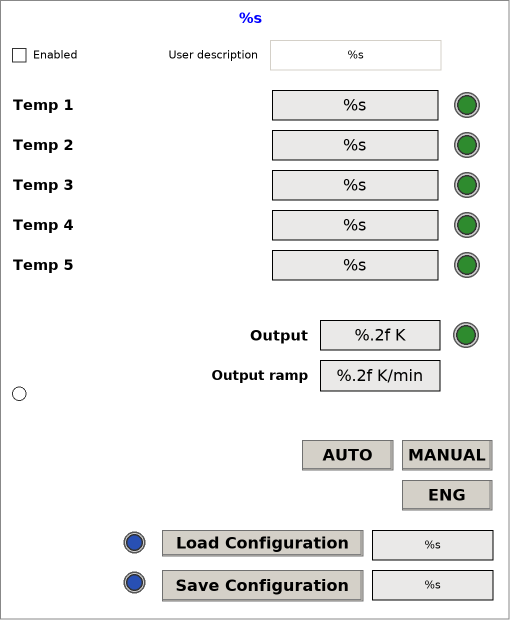
VISUALIZATION TEMPLATE_TEMPERATURE_VOTE  // 510x620
VAR_IN_OUT
	m_Instance : FB_METIS_VOTER; 
	m_all_temperatures_array: FB_METIS_TEMPERATURES;
END_VAR
    Rectangle (10,3 481x30), "%s", tooltip "vote Temperature", text variable: m_Instance.in_sName
    Rectangle (10,90 68x30), "Temp 1"
    Rectangle (10,130 68x30), "Temp 2"
    Rectangle (10,170 68x30), "Temp 3"
    Rectangle (10,210 68x30), "Temp 4"
    Rectangle (10,250 68x30), "Temp 5"
    Lamp1 (452,90 30x30), variable: m_Instance.aTempPointers[0]^.stat.bValid, style: Lamp-Lamp1-Green
    Lamp1 (452,130 30x30), variable: m_Instance.aTempPointers[1]^.stat.bValid, style: Lamp-Lamp1-Green
    Lamp1 (452,170 30x30), variable: m_Instance.aTempPointers[2]^.stat.bValid, style: Lamp-Lamp1-Green
    Lamp1 (452,210 30x30), variable: m_Instance.aTempPointers[3]^.stat.bValid, style: Lamp-Lamp1-Green
    Lamp1 (452,250 30x30), variable: m_Instance.aTempPointers[4]^.stat.bValid, style: Lamp-Lamp1-Green
    RadioButton (10,306 162x175), variable: m_Instance.stat.nVoteMethod, input disabled if: NOT m_Instance.bEngMode
        Areas[0]: Text=Lowest Temperature
        Areas[1]: Text=Highest Temperature
        Areas[2]: Text=Average
        Areas[3]: Text=First Valid
        p340057476: Lowest Temperature
        p3123465237: Highest Temperature
        p2481256679: Average
        p1032612214: First Valid
        p3228930307: Median
        p1847394450: Temperature 2oo3
        p1205187680: Temperature 3oo5
    Rectangle (320,320 120x30), "%.2f K", tooltip "Voting Temperature out [K]", text variable: m_instance.stat.lrTempK
    Lamp1 (451,320 30x30), variable: m_Instance.stat.bValid, style: Lamp-Lamp1-Green
    Rectangle (272,90 166x30), "%s", tooltip "Voting Temperature out [K]", text variable: m_Instance.aTempPointers[0]^.stat.sName
    Rectangle (272,130 166x30), "%s", tooltip "Voting Temperature out [K]", text variable: m_Instance.aTempPointers[1]^.stat.sName
    Rectangle (272,170 166x30), "%s", tooltip "Voting Temperature out [K]", text variable: m_Instance.aTempPointers[2]^.stat.sName
    Rectangle (272,210 166x30), "%s", tooltip "Voting Temperature out [K]", text variable: m_Instance.aTempPointers[3]^.stat.sName
    Rectangle (272,250 166x30), "%s", tooltip "Voting Temperature out [K]", text variable: m_Instance.aTempPointers[4]^.stat.sName
    Button (302,440 91x30), "AUTO", tooltip "Switch to AUTO Mode", colour toggle: m_instance.bAutoMode, input disabled if: m_instance.bAutoMode OR m_instance.bEngMode
        OnMouseClick: execute { m_instance.bAutoMode := TRUE; m_instance.bPLC_HMI := FALSE; }
    Button (402,480 90x30), "ENG", tooltip "Toggle Engineering Mode", colour toggle: m_instance.bEngMode, input disabled if: m_instance.bAutoMode
        toggle m_instance.bEngMode
    Button (402,440 90x30), "MANUAL", tooltip "Switch to MANUAL Mode", colour toggle: NOT m_instance.bAutoMode, input disabled if: NOT m_instance.bAutoMode AND NOT m_instance.bEngMode
        OnMouseClick: execute {
            m_instance.bAutoMode := FALSE;
            m_instance.bManualMode := TRUE;
            m_instance.bPLC_HMI := TRUE;
        }
    Lamp1 (122,530 25x25), tooltip "Command coming from the Control System", variable: m_instance.bReadConfig, style: Lamp-Lamp1-Blue
    Button (162,570 201x31), "Save Configuration", input disabled if: NOT m_instance.bEngMode
        OnMouseClick: execute { m_instance.bWriteConfig := TRUE; }
    Button (162,530 201x26), "Load Configuration", input disabled if: NOT m_instance.bEngMode
        OnMouseClick: execute { m_instance.bReadConfig := TRUE; }
    Lamp1 (122,570 25x25), tooltip "Command coming from the Control System", variable: m_instance.bWriteConfig, style: Lamp-Lamp1-Blue
    Rectangle (320,360 120x31), "%.2f K/min", tooltip "Ramp [K/min]", text variable: m_instance.stat.lrRamp
    Rectangle (372,530 121x30), "%s", text variable: m_Instance.fbTempVoteConfig.sReadError, colour toggle: m_Instance.fbTempVoteConfig.bReadError
    Rectangle (372,570 121x30), "%s", text variable: m_Instance.fbTempVoteConfig.sWriteError, colour toggle: m_Instance.fbTempVoteConfig.bWriteError
    Checkbox (10,40 111x30), "Enabled", variable: m_Instance.stat.bEnabled, input disabled if: NOT m_Instance.bEngMode
    Label (110,40 151x30), "User description"
    Textfield (270,40 171x30), "%s", text variable: m_Instance.stat.sDescription, input disabled if: NOT m_Instance.bEngMode
        OnMouseClick: write the text variable via Default
    Rectangle (210,320 101x31), "Output"
    Rectangle (210,360 101x31), "Output ramp"
END_VISUALIZATION

// HMI/VISUs/Util/Button/VISU_HMI_ROUTINES_BUTTON
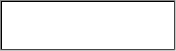
VISUALIZATION VISU_HMI_ROUTINES_BUTTON  // 176x51
VAR_IN_OUT
    m_Hmi : FB_HMI_BUTTON;
END_VAR
    Rectangle (0,0 175x50), invisible if: m_Hmi.bIsNotOrange
    Rectangle (0,0 175x50), invisible if: m_Hmi.bIsNotGray
    Rectangle (0,0 175x50), invisible if: m_Hmi.bIsNotBlue
    Rectangle (0,0 175x50), invisible if: m_Hmi.bIsNotRed
    Rectangle (0,0 175x50), invisible if: m_Hmi.bIsNotGreen
    Rectangle (0,0 175x50), "%s", text variable: m_Hmi.sName
    Rectangle (0,0 175x50), invisible if: m_Hmi.bNotActivated
    Line (0,49) (175,49), invisible if: m_Hmi.bActivated
    Line (174,0) (174,50), invisible if: m_Hmi.bActivated
    Line (174,0) (0,0), invisible if: m_Hmi.bActivated
    Line (0,49) (0,0), invisible if: m_Hmi.bActivated
    Line (175,50) (175,1), invisible if: m_Hmi.bNotActivated
    Line (0,1) (174,1), invisible if: m_Hmi.bNotActivated
    Line (1,0) (1,49), invisible if: m_Hmi.bNotActivated
    Line (175,50) (1,50), invisible if: m_Hmi.bNotActivated
END_VISUALIZATION

// HMI/VISUs/Util/Button/VISU_HMI_SUBSUBSYSTEM_BUTTON
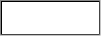
VISUALIZATION VISU_HMI_SUBSUBSYSTEM_BUTTON  // 101x36
VAR_IN_OUT
    m_Hmi : FB_HMI_BUTTON;
END_VAR
    Rectangle (0,0 100x35), invisible if: m_Hmi.bIsNotOrange
    Rectangle (0,0 100x35), invisible if: m_Hmi.bIsNotGray
    Rectangle (0,0 100x35), invisible if: m_Hmi.bIsNotBlue
    Rectangle (0,0 100x35), invisible if: m_Hmi.bIsNotRed
    Rectangle (0,0 100x35), invisible if: m_Hmi.bIsNotGreen
    Rectangle (0,0 100x35), "%s", text variable: m_Hmi.sName
    Rectangle (0,0 100x35), invisible if: m_Hmi.bNotActivated
    Line (0,34) (100,34), invisible if: m_Hmi.bActivated
    Line (99,0) (99,35), invisible if: m_Hmi.bActivated
    Line (98,0) (0,0), invisible if: m_Hmi.bActivated
    Line (0,35) (0,0), invisible if: m_Hmi.bActivated
    Line (100,35) (100,1), invisible if: m_Hmi.bNotActivated
    Line (0,1) (99,1), invisible if: m_Hmi.bNotActivated
    Line (1,0) (1,35), invisible if: m_Hmi.bNotActivated
    Line (100,35) (1,35), invisible if: m_Hmi.bNotActivated
END_VISUALIZATION

// HMI/VISUs/Util/Button/VISU_HMI_SUBSYSTEM_BUTTON
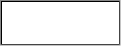
VISUALIZATION VISU_HMI_SUBSYSTEM_BUTTON  // 121x46
VAR_IN_OUT
    m_Hmi : FB_HMI_BUTTON;
END_VAR
    Rectangle (0,0 120x45), invisible if: m_Hmi.bIsNotOrange
    Rectangle (0,0 120x45), invisible if: m_Hmi.bIsNotGray
    Rectangle (0,0 120x45), invisible if: m_Hmi.bIsNotBlue
    Rectangle (0,0 120x45), invisible if: m_Hmi.bIsNotRed
    Rectangle (0,0 120x45), invisible if: m_Hmi.bIsNotGreen
    Rectangle (0,0 120x45), "%s", text variable: m_Hmi.sName
    Rectangle (0,0 120x45), invisible if: m_Hmi.bNotActivated
    Line (0,44) (120,44), invisible if: m_Hmi.bActivated
    Line (119,0) (119,45), invisible if: m_Hmi.bActivated
    Line (118,0) (0,0), invisible if: m_Hmi.bActivated
    Line (0,45) (0,0), invisible if: m_Hmi.bActivated
    Line (120,45) (120,1), invisible if: m_Hmi.bNotActivated
    Line (0,1) (119,1), invisible if: m_Hmi.bNotActivated
    Line (1,0) (1,45), invisible if: m_Hmi.bNotActivated
    Line (120,45) (1,45), invisible if: m_Hmi.bNotActivated
END_VISUALIZATION

// HMI/VISUs/Util/Button/VISU_HMI_SYSTEM_BUTTON
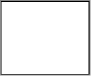
VISUALIZATION VISU_HMI_SYSTEM_BUTTON  // 91x76
VAR_IN_OUT
    m_Hmi : FB_HMI_BUTTON;
END_VAR
    Rectangle (0,0 90x75), invisible if: m_Hmi.bIsNotOrange
    Rectangle (0,0 90x75), invisible if: m_Hmi.bIsNotGray
    Rectangle (0,0 90x75), invisible if: m_Hmi.bIsNotBlue
    Rectangle (0,0 90x75), invisible if: m_Hmi.bIsNotRed
    Rectangle (0,0 90x75), invisible if: m_Hmi.bIsNotGreen
    Rectangle (0,50 90x25), "%s", text variable: m_Hmi.sName
    Image (25,10 40x40), image: VISU_HMI_BUTTON_IMAGES.Start
        p84334746: m_Hmi.sIconName
    Rectangle (0,0 90x75), invisible if: m_Hmi.bNotActivated
    Line (0,74) (90,74), invisible if: m_Hmi.bActivated
    Line (89,75) (89,0), invisible if: m_Hmi.bActivated
    Line (0,74) (0,0), invisible if: m_Hmi.bActivated
    Line (88,0) (0,0), invisible if: m_Hmi.bActivated
    Line (0,1) (90,1), invisible if: m_Hmi.bNotActivated
    Line (1,75) (1,0), invisible if: m_Hmi.bNotActivated
    Line (90,75) (1,75), invisible if: m_Hmi.bNotActivated
    Line (90,75) (90,1), invisible if: m_Hmi.bNotActivated
END_VISUALIZATION

// HMI/VISU_HMI
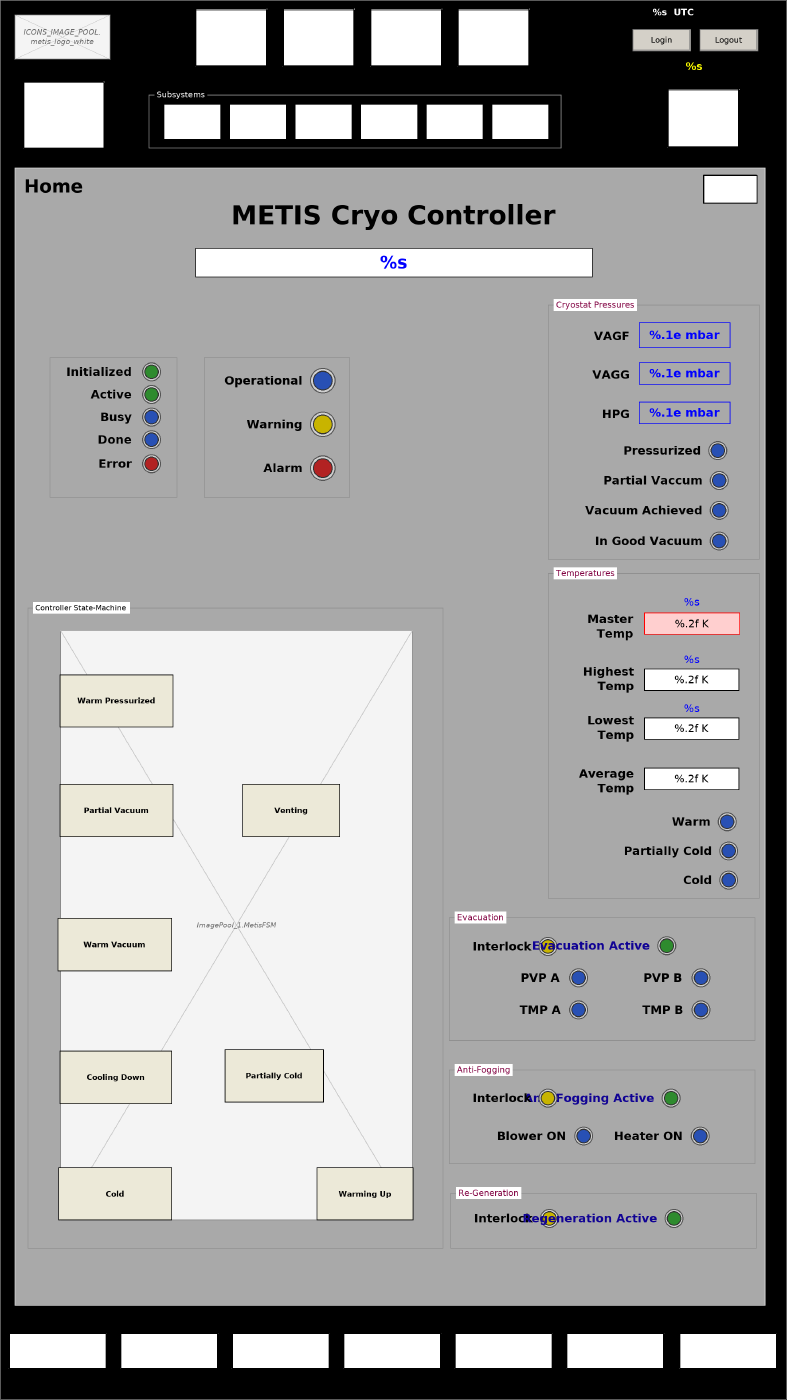
VISUALIZATION VISU_HMI  // 1080x1920
    Frame (388,12 100x80)
        shows VISU_HMI_SYSTEM_BUTTON(m_Hmi := PRG_HMI.fbServicesButton)
        OnMouseClick: execute { PRG_HMI.eActiveTab := E_HMI_TABS.SERVICES; }
    Frame (268,12 100x80)
        shows VISU_HMI_SYSTEM_BUTTON(m_Hmi := PRG_HMI.fbHomeButton)
        OnMouseClick: execute { PRG_HMI.eActiveTab := E_HMI_TABS.HOME; }
    Rectangle (20,230 1030x1560)
    Frame (20,230 1030x1560), frame switch variable: PRG_HMI.eActiveTab
        shows VISU_HMI_HOME(m_instance := MAIN.met_cryo_ctrl)
        shows VISU_HMI_SERVICES()
        shows VISU_HMI_EVACUATION()
        shows VISU_HMI_COOL_DOWN(m_instance := MAIN.met_cryo_ctrl.met_cool_down, m_Cry_Instance := MAIN.met_cryo_ctrl)
        shows VISU_HMI_WARM_UP(m_instance := MAIN.met_cryo_ctrl.met_warm_up, m_Cry_Instance := MAIN.met_cryo_ctrl)
        shows VISU_HMI_VENTING(m_instance := MAIN.met_cryo_ctrl.met_venting, m_Cry_Instance := MAIN.met_cryo_ctrl)
        shows VISU_HMI_ANTI_FOGGING(m_instance := MAIN.met_cryo_ctrl.met_anti_fogging)
        shows VISU_HMI_REGENERATION(m_instance := MAIN.met_cryo_ctrl.met_regeneration)
        shows VISU_HMI_POWER_OUTAGE()
        shows VISU_HMI_CABINETS()
        shows VISU_HMI_VALVES()
        shows VISU_HMI_CONTROL_UNITS()
        shows VISU_HMI_CRY(met_cryo_ctrl := MAIN.met_cryo_ctrl, m_Hmi := PRG_HMI.fbCry)
        shows VISU_HMI_CFO()
        shows VISU_HMI_IMG(m_Temperatures := MAIN.met_cryo_ctrl.met_temp, m_Voters := MAIN.met_cryo_ctrl.met_voters, m_Tctrl := MAIN.met_cryo_ctrl.met_tctrl, m_Heaters := MAIN.met_cryo_ctrl.met_heaters, m_Lakeshores := MAIN.met_cryo_ctrl.met_lakeshores, m_Hmi := PRG_HMI.fbImg)
        shows VISU_HMI_LMS()
        shows VISU_HMI_SCA(m_Temperatures := MAIN.met_cryo_ctrl.met_temp, m_Voters := MAIN.met_cryo_ctrl.met_voters, m_Tctrl := MAIN.met_cryo_ctrl.met_tctrl, m_Heaters := MAIN.met_cryo_ctrl.met_heaters, m_Lakeshores := MAIN.met_cryo_ctrl.met_lakeshores, m_Hmi := PRG_HMI.fbSca)
        shows VISU_HMI_ICS(m_CCUs := MAIN.met_cryo_ctrl.met_ccus, m_Hmi := PRG_HMI.fbIcs)
        shows VISU_HMI_HEATERS()
        shows VISU_HMI_EVENTS()
        shows VISU_HMI_PRESSURES()
        shows VISU_HMI_COOLERS()
        shows VISU_HMI_PUMPS(m_Hmi := PRG_HMI.fbPumps)
        shows VISU_HMI_TEMPERATURES(met_cryo_ctrl := MAIN.met_cryo_ctrl, m_Hmi := PRG_HMI.fbTemperatures)
        shows VISU_HMI_ICS_INTERLOCKS()
        shows VISU_HMI_DETECTORS()
        shows VISU_HMI_CONTROL_LOOPS()
        shows VISU_SIM_PRESS_AND_TEMPS()
        pReferences[1]: m_Instance=MAIN.fbServices, m_Hmi=PRG_HMI.fbServices
        p1199675002: PRG_HMI.fbSca
        p3123483648: PRG_HMI.fbPumps
        p2939190159: MAIN.met_cryo_ctrl
    Image (20,20 131x61), image: ICONS_IMAGE_POOL.metis_logo_white
    Rectangle (774,4 300x25), "%s UTC", text variable: MAIN.met_cryo_ctrl.met_cry_time.stat.sUtcTime
    Frame (12,1828 135x50)
        shows VISU_HMI_ROUTINES_BUTTON(m_Hmi := PRG_HMI.fbEvacuationButton)
        OnMouseClick: execute { PRG_HMI.eActiveTab := E_HMI_TABS.EVACUATION; }
    Frame (165,1828 135x50)
        shows VISU_HMI_ROUTINES_BUTTON(m_Hmi := PRG_HMI.fbCoolDownButton)
        OnMouseClick: execute { PRG_HMI.eActiveTab := E_HMI_TABS.COOL_DOWN; }
    Frame (318,1828 135x50)
        shows VISU_HMI_ROUTINES_BUTTON(m_Hmi := PRG_HMI.fbWarmUpButton)
        OnMouseClick: execute { PRG_HMI.eActiveTab := E_HMI_TABS.WARM_UP; }
    Frame (471,1828 135x50)
        shows VISU_HMI_ROUTINES_BUTTON(m_Hmi := PRG_HMI.fbVentingButton)
        OnMouseClick: execute { PRG_HMI.eActiveTab := E_HMI_TABS.VENTING; }
    Frame (624,1828 135x50)
        shows VISU_HMI_ROUTINES_BUTTON(m_Hmi := PRG_HMI.fbRegenerationButton)
        OnMouseClick: execute { PRG_HMI.eActiveTab := E_HMI_TABS.REGENERATION; }
    Frame (777,1828 135x50)
        shows VISU_HMI_ROUTINES_BUTTON(m_Hmi := PRG_HMI.fbAntiFoggingButton)
        OnMouseClick: execute { PRG_HMI.eActiveTab := E_HMI_TABS.ANTI_FOGGING; }
    Frame (932,1828 135x50)
        shows VISU_HMI_ROUTINES_BUTTON(m_Hmi := PRG_HMI.fbPowerOutageButton)
        OnMouseClick: execute { PRG_HMI.eActiveTab := E_HMI_TABS.POWER_OUTAGE; }
    Frame (508,12 100x80)
        shows VISU_HMI_SYSTEM_BUTTON(m_Hmi := PRG_HMI.fbEventsButton)
        OnMouseClick: execute { PRG_HMI.eActiveTab := E_HMI_TABS.EVENTS; }
    Frame (628,12 100x80)
        shows VISU_HMI_SYSTEM_BUTTON(m_Hmi := PRG_HMI.fbIcsInterlocksButton)
        OnMouseClick: execute { PRG_HMI.eActiveTab := E_HMI_TABS.ICS_INTERLOCKS; }
    GroupBox (204,122 566x81), "Subsystems"
        Frame (20,20 80x51)
            shows VISU_HMI_SUBSYSTEM_BUTTON(m_Hmi := PRG_HMI.fbCryButton)
            OnMouseClick: execute { PRG_HMI.eActiveTab := E_HMI_TABS.SUBSYSTEMS_CRY; }
        Frame (110,20 80x51)
            shows VISU_HMI_SUBSYSTEM_BUTTON(m_Hmi := PRG_HMI.fbCfoButton)
            OnMouseClick: execute { PRG_HMI.eActiveTab := E_HMI_TABS.SUBSYSTEMS_CFO; }
        Frame (200,20 80x51)
            shows VISU_HMI_SUBSYSTEM_BUTTON(m_Hmi := PRG_HMI.fbImgButton)
            OnMouseClick: execute { PRG_HMI.eActiveTab := E_HMI_TABS.SUBSYSTEMS_IMG; }
        Frame (290,20 80x51)
            shows VISU_HMI_SUBSYSTEM_BUTTON(m_Hmi := PRG_HMI.fbLmsButton)
            OnMouseClick: execute { PRG_HMI.eActiveTab := E_HMI_TABS.SUBSYSTEMS_LMS; }
        Frame (380,20 80x51)
            shows VISU_HMI_SUBSYSTEM_BUTTON(m_Hmi := PRG_HMI.fbScaButton)
            OnMouseClick: execute { PRG_HMI.eActiveTab := E_HMI_TABS.SUBSYSTEMS_SCA; }
        Frame (470,20 80x51)
            shows VISU_HMI_SUBSYSTEM_BUTTON(m_Hmi := PRG_HMI.fbIcsButton)
            OnMouseClick: execute { PRG_HMI.eActiveTab := E_HMI_TABS.SUBSYSTEMS_ICS; }
    Group (868,40 172x66)
        Button (0,0 80x30), "Login"
            OnMouseClick:  Type=Login, OpenCentered=True
        Button (92,0 80x30), "Logout"
            OnMouseClick:  Type=Logout, OpenCentered=True
        Rectangle (0,36 169x30), "%s", tooltip "Current user", text variable: MAIN.met_cryo_ctrl.current_user
    Frame (916,122 100x81)
        shows VISU_HMI_SYSTEM_BUTTON(m_Hmi := PRG_HMI.fbDevicesButton)
        OnMouseClick:  Dialog=VISU_HMI_DEVICES_DIALOG, OpenModal=True, PositionX=856, PositionY=228
    Frame (32,112 113x93), invisible if: NOT MAIN.met_cryo_ctrl.stat.bSimulation
        shows VISU_HMI_SYSTEM_BUTTON(m_Hmi := PRG_HMI.fbCryoSimButton)
        OnMouseClick: execute { PRG_HMI.eActiveTab := E_HMI_TABS.SIMULATION; }
END_VISUALIZATION

(* text list TEXTLIST_METIS_CTRL_MODE (id | default)
  1 | Auto
  2 | Manual
   |  *)
